FUNCTION_BLOCK FB_RANDOM (* Generate a REAL Randomly *)
  (* Standard: 61499-1; Classification: Mathematic; Function: RANDOM; Type: Mathematical function; Description: Copyright (c) 2012 Profactor GmbH This program and the accompanying materials are made available under the terms of the Eclipse Public License 2.0 which is available at https://www.eclipse.org/legal/epl-2.0/ SPDX-License-Identifier: EPL-2.0 *)
  (* Version 3.0, 2025-04-14, Patrick Aigner, changed package *)
  (* Version 1.0, 2012-05-31, Gerhard Ebenhofer, Profactor GmbH *)
  PACKAGE eclipse4diac::utils;
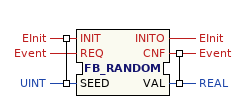
  EVENT_INPUT
    INIT : EInit WITH SEED; (* Initializes the random with the specified seed, if not called the generated values will always be identical *)
    REQ; (* Calculates a new random number between 0 and 1 *)
  END_EVENT
  EVENT_OUTPUT
    INITO : EInit;
    CNF WITH VAL; (* Execution Confirmation *)
  END_EVENT
  VAR_INPUT
    SEED : UINT := 0; (* the seed to initialize the random, a seed of 0 (zero) uses the current systemtime as seed *)
  END_VAR
  VAR_OUTPUT
    VAL : REAL; (* Function output *)
  END_VAR
END_FUNCTION_BLOCK
